FUNCTION_BLOCK TmsEmbarkSingleSwitch EXTENDS Process IMPLEMENTS ITF_SwitchStation
VAR
	DepartMover : I_XtsMover;
	ExecuteSequence : BOOL;
	Axis : AXIS_REF;
	SwitchAxis : Axis_Base(Axis);
	_switchLoadPosition : MC_LREAL;
	_switchUnloadPosition : MC_LREAL;
	State :(
		Init,                                               
		Ready,                                 
        Waiting,
		HasSwitch,
		Boarding,
		BoardingComplete,
		Moving,
		ActivateTrackForMover,
		CheckTrackActive,
		ReturnHome,
		Done,
		Aborting); 
	_switchPosition: MC_LREAL;
	_TargetTrackId : I_XtsTrack;
	_BoardVelocity : MC_LREAL;
	_SwitchVelocity : MC_LREAL;
END_VAR

PROPERTY BoardVelocity : MC_LREAL
GET
BoardVelocity := _BoardVelocity;
END_GET
SET
_BoardVelocity := BoardVelocity;
END_SET
END_PROPERTY

METHOD PUBLIC  Cycle : HRESULT
VAR
	ActivateTrackResult : BOOL;
	BoardMoverResult : HRESULT;
	BaseCallResult : HRESULT;
END_VAR
Cycle := S_OK;
CASE State OF
	Init:
		_Operating := _Empty := _Complete := _Ready := _HasMover := FALSE;
		StationMovers := 0;
		State := Ready;
	
	Ready:	
		IF ExecuteSequence THEN
			_Operating := _Complete := _HasMover := FALSE;
			_Empty := _Ready := TRUE;
			StationMovers := 0;
			State := Waiting;
		END_IF
	
	Waiting:
		IF _HasMover THEN
			State := HasSwitch;
			_Operating := TRUE;
			_Empty := FALSE;
			_Ready := FALSE;
			_Complete := FALSE;
		END_IF
	
	HasSwitch:
		IF SwitchAxis.isAtPosition(position := _switchLoadPosition) THEN
			State := Boarding;
		END_IF
			
	Boarding:
		BoardMoverResult := DepartMover.MoveTo(RequiredPosition := _switchPosition, MoveVelocity := _BoardVelocity, NonModuloMove := TRUE);
		IF DepartMover.isMoverAtPosition(position := _switchPosition) THEN
			State := BoardingComplete;
		END_IF
		
	BoardingComplete:
		IF Succeeded( SwitchAxis.MoveToPosition(Position := _switchUnloadPosition, Velocity := _SwitchVelocity)) THEN
			State := Moving;
		END_IF
		
	Moving:
		IF NOT SwitchAxis.isStationary() THEN
			State := ActivateTrackForMover;
		END_IF
		
	ActivateTrackForMover:
		DepartMover.ActivateTrack(NewTrack := _TargetTrackId.MyOTCID,Track := _TargetTrackId);		
		State := CheckTrackActive;

	CheckTrackActive:
		IF DepartMover.MoversActiveTrack = _TargetTrackId.MyOTCID AND SwitchAxis.isAtPosition(position := _switchUnloadPosition) THEN
			State := ReturnHome;
			_Complete := TRUE;
		END_IF
	
	ReturnHome:
		IF SUCCEEDED( SwitchAxis.MoveToPosition(Position := _switchLoadPosition, Velocity := _SwitchVelocity)) THEN
			State := Done;
		END_IF
			
	Done:
		IF _Complete AND NOT _HasMover THEN
			_Operating := FALSE;
			_Empty := TRUE;
			_Ready := TRUE;
			State := Waiting;
		END_IF

	Aborting:
		State := Ready;	
		DepartMover := 0;
	ELSE
		Cycle := E_FAIL;
END_CASE
BaseCallResult := SUPER^.Cycle();
SwitchAxis.Cycle();
END_METHOD

METHOD DisableLift : HRESULT
VAR_INPUT
END_VAR
SwitchAxis.DisableAxis();
END_METHOD

METHOD EnableLift : HRESULT
VAR_INPUT
END_VAR
SwitchAxis.EnableAxis(FALSE,FALSE);
END_METHOD

METHOD HasMover : BOOL
VAR_INPUT
	mover : I_XtsMover;
END_VAR
IF StationMovers <= 2 THEN
	StationMovers := StationMovers + 1;
	DepartMover := mover;
	_HasMover := TRUE;
END_IF
HasMover := TRUE;
END_METHOD

METHOD PUBLIC MoverAway : BOOL
VAR_INPUT
END_VAR
StationMovers := StationMovers - 1;
IF StationMovers = 0 THEN
	_HasMover := FALSE;
END_IF
DepartMover := 0;
MoverAway := TRUE;
END_METHOD

METHOD ResetLift : HRESULT
VAR_INPUT
END_VAR
SwitchAxis.Reset();
END_METHOD

METHOD StartSwitch : BOOL
VAR_INPUT
END_VAR
ExecuteSequence := true;
END_METHOD

METHOD StopSwitch : BOOL
VAR_INPUT
END_VAR
ExecuteSequence := FALSE;
State := Aborting;
END_METHOD

PROPERTY SwitchLoadPosition : MC_LREAL
GET
SwitchLoadPosition := _switchLoadPosition;
END_GET
SET
_switchLoadPosition := SwitchLoadPosition;
END_SET
END_PROPERTY

METHOD SwitchMoveComplete : BOOL
END_METHOD

PROPERTY SwitchTravelPosition : mc_lreal
GET
SwitchTravelPosition := _switchPosition;
END_GET
SET
_switchPosition := SwitchTravelPosition;
END_SET
END_PROPERTY

PROPERTY SwitchUnloadPosition : MC_LREAL
GET
SwitchUnloadPosition := _switchUnloadPosition;
END_GET
SET
_switchUnloadPosition := SwitchUnloadPosition;
END_SET
END_PROPERTY

PROPERTY SwitchVelocity : MC_LREAL
GET
SwitchVelocity := _SwitchVelocity;
END_GET
SET
_SwitchVelocity := SwitchVelocity;
END_SET
END_PROPERTY

PROPERTY TargetTrackId : I_XtsTrack
GET
TargetTrackId := _TargetTrackId;
END_GET
SET
_TargetTrackId := TargetTrackId;
END_SET
END_PROPERTY

END_FUNCTION_BLOCK

(* stored: Version 1.1.0.1
   POU TmsEmbarkSingleSwitch: Id {a1345a8f-d28a-4176-804e-11454f70b667}, SpecialFunc None
   Property BoardVelocity: Id {831e3c6b-034b-4353-83d0-e3165e0635f3}
   Get Get: Id {29602b3a-b998-4746-b889-c90549b64635}
   Set Set: Id {2fe6cf87-3d91-4f0d-abae-291448af5dcf}
   Method Cycle: Id {992aa554-6501-4e8f-af38-b1f2b991a987}
   Method DisableLift: Id {48178ec4-8b43-421e-9fb5-b7445276f569}
   Method EnableLift: Id {50ffe6bd-500f-4895-ac7f-2f448330de69}
   Method HasMover: Id {3dfbfe5d-88fb-42cd-8ef4-33bfd88b9fd1}
   Method MoverAway: Id {e0f828f0-4af6-4c6b-903d-ca5a359a945a}
   Method ResetLift: Id {e01d8d04-17e3-496e-b671-f1b1ca8fff28}
   Method StartSwitch: Id {ae2b2fa3-2884-439d-8324-d04aeee3d2a6}
   Method StopSwitch: Id {cac109d7-36fe-4bcd-8860-a58bd7cdbe98}
   Property SwitchLoadPosition: Id {8a954b15-9e2e-45e2-9983-586f0bb0d4ea}
   Get Get: Id {c7c8f444-a876-46f4-b0cb-0dad5a2a0e8f}
   Set Set: Id {53f3e315-b71d-472a-98ca-6f0d73523ae9}
   Method SwitchMoveComplete: Id {5e3f9db3-9a4d-4699-9458-649b47840420}
   Property SwitchTravelPosition: Id {56005ce1-5a9a-45b9-af03-9875bac9d76b}
   Get Get: Id {9d4f14ba-9356-4943-857d-bfbb12a15568}
   Set Set: Id {041c3047-5928-4394-9507-73b44fee711b}
   Property SwitchUnloadPosition: Id {6faedafb-b954-46db-8550-5042a177e286}
   Get Get: Id {8d3d0655-9fc3-4248-beaa-e60d661cc7f6}
   Set Set: Id {da277918-2a30-4cfc-8615-b9ef5ee09b08}
   Property SwitchVelocity: Id {5bee5216-580a-4c92-a98e-135910f268ec}
   Get Get: Id {5f6d59ad-16e2-4d95-8537-c0fe3c94515a}
   Set Set: Id {9a50fe25-bba9-43bc-969b-72a95486a8df}
   Property TargetTrackId: Id {60f84ea8-30a8-4877-b5ee-78b5070ad98e}
   Get Get: Id {cbe6c8be-4cbe-4755-ac3d-aca3acacdfc2}
   Set Set: Id {1aa8ea54-81af-46d8-bdb2-7bd4b3a74fb9} *)
